TYPE ST_CFG_Subsystem :
(**************************************************************************************
 * 	Application		:	BoxControl Framework
 *	Revision		:	$Revision: 404529 $
 *	Revision date	:	$Date: 2018-04-23 08:21:38 +0200 (Mo., 23 Apr 2018) $
 *	Last changed by	:	$Author: b7bolm $
 *	URL				:	$URL: http://almscdc.swisslog.com/repo/SWPD/Development/BoxControlFramework/20_Release/trunk/01_Software/BCF/BCF/JumpStart/20_Product/10_App/15_Subsystem/10_Lib/10_Conv/01_DUTs/10_Dummy/ST_CFG_Subsystem.TcDUT $
 *
 *	Purpose			:	Subsystem configuration
 *
 * ------------------------------------------------------------------------------------
 *	Copyright Swisslog [IP AG], Switzerland. All rights reserved.
 * 
 * ------------------------------------------------------------------------------------
 *	
 * 	Revision History: 
 *
 * 	VERSION			DATE			INITIALS			DESCRIPTION
 *	0.1				01.01.2001		swl					Example
 *
 **************************************************************************************)
STRUCT
	SubsystemName				: STRING(NAME_LENGTH); // Name of the Subsystem 
	SubsystemNumber				: INT; // Number of the Subsystem 
	MaxInitCallsPerCycle		: INT; // Maximum of initialization calls in one cycle
	MinMasterSpeed				: INT; // Min master speed [%]
	MaxMasterSpeed				: INT; // Max master speed [%]
END_STRUCT
END_TYPE

(* stored: Version 1.1.0.1, ProductVersion 3.1.4022.12
   DUT ST_CFG_Subsystem: Id {85e6bcfc-96f5-4d81-b9cb-9fdc14abaf48} *)
